// modulo (shortest way)/absolute movements
// -- - + ++
// move / pos / velo
// stop / reset
TYPE ST_AxisControlManual :
STRUCT
	bEnable										: BOOL;
	bModulo										: BOOL;
	bSlowForward								: BOOL;
	bSlowBackward								: BOOL;
	bFastForward								: BOOL;
	bFastBackward								: BOOL;
	bStop										: BOOL;
	bReset										: BOOL;
	bExecute									: BOOL;
	fVelocity									: LREAL;
	fPosition									: LREAL;
	fOverride									: LREAL;
END_STRUCT
END_TYPE

(* stored: Version 1.2.0.0, ProductVersion 3.1.4026.13, FileIdentifier 701615645f85904552f4347f0cdb90181d145d88, FileSignature 90b93b1500d6f0be20f8cd1b7edcbe4a2caf7e47b5dde88d3eb40320650680994b3e103bac8580e5acb61927b3f0b2e243efa0c7dd873389b477525103840cd825249d9d0202967f7b52804452ca950ff7ae829d73f1aa56f1d61350e7c625a803447868d33d9289bbd268cf0cc93d41d39ebe2ab1f49ed802da07f942d4806364036ca50d7e764e54f8e19b550d47f203a7b337a78940b1b9dc8e0c05b9fd59f58f88a02ed96d6e4919fb3f5ac071514ee35bbcd03f8b07fdd8380cbbb7596bc598231ed27aa138a78025d361574e8ef4b030d9324978cdf5066724afb402c07ee91a4477ac8bcf242b74aaf146cf1fd05a177639c76348e5d5df08823c3377
   DUT ST_AxisControlManual: Id {bd6b0ac2-380f-4722-9a14-1a09383174fe} *)
